{attribute addProperty BoxType "ELX3252-0000-0016"}
{attribute addProperty Id "Limit_1_BIT_0BIT10.1253Limit_1_BIT_1BIT10.1253Limit_2_BIT_0BIT10.1255Limit_2_BIT_1BIT10.1255ErrorBIT10.1257TxPDO_StateBIT10.12515TxPDO_ToggleBIT10.12516"}
{attribute addProperty CRC "1930103016"}
{attribute addProperty SizeInBites "16"}
{attribute addProperty SizeInBytes "2"}
TYPE Status_730B08E8 :
STRUCT
	{attribute 'hide'}
	reserve_1_BIT_0 : BIT;
	{attribute 'hide'}
	reserve_1_BIT_1 : BIT;
	{attribute addProperty Name "Limit_1"}
	Limit_1_BIT_0 : BIT;
	{attribute addProperty Name "Limit_1"}
	Limit_1_BIT_1 : BIT;
	{attribute addProperty Name "Limit_2"}
	Limit_2_BIT_0 : BIT;
	{attribute addProperty Name "Limit_2"}
	Limit_2_BIT_1 : BIT;
	{attribute addProperty Name "Error"}
	Error : BIT;
	{attribute 'hide'}
	reserve_2 : BIT;
	{attribute 'hide'}
	reserve_3_BIT_0 : BIT;
	{attribute 'hide'}
	reserve_3_BIT_1 : BIT;
	{attribute 'hide'}
	reserve_3_BIT_2 : BIT;
	{attribute 'hide'}
	reserve_3_BIT_3 : BIT;
	{attribute 'hide'}
	reserve_3_BIT_4 : BIT;
	{attribute 'hide'}
	reserve_3_BIT_5 : BIT;
	{attribute addProperty Name "TxPDO_State"}
	TxPDO_State : BIT;
	{attribute addProperty Name "TxPDO_Toggle"}
	TxPDO_Toggle : BIT;
END_STRUCT
END_TYPE

(* stored: Version 1.2.0.0, ProductVersion 3.1.4024.9
   DUT Status_730B08E8: Id {97272974-b47c-4162-921b-2691df19e634} *)
